FUNCTION_BLOCK AR_CALIBRATE_3P_REF (* Adapter-based 3-point calibration for joysticks/sensors with a center position (Min, Mid, Max), free order like AR_CALIBRATE_3P - reference targets (Y_MIN/Y_MID/Y_MAX) are live AR sockets, persisted via 3 additional AR2 plugs (MIN_REF/MID_REF/MAX_REF), same live-echo pattern as AR_CALIBRATE_SQ_REF/AR_CALIBRATE_2P_REF *)
  (* Standard: 61499-1 *)
  (* Version 1.0, 2026-09-11, Meisterschulen am Ostbahnhof, 3-Punkt-Pendant zu AR_CALIBRATE_2P_REF - fuer Sensoren mit definierter Mittelstellung (z.B. Lenkwinkelsensor: links/geradeaus/rechts). Keine ECC-Reihenfolge-Erzwingung: C_MIN/C_MID/C_MAX speichern unabhaengig, wie AR_CALIBRATE_3P. *)
  (* Version 1.3, 2026-09-21, Franz Höpfinger, Code-Review-Fund (PR #260): xClipping clippte bisher unconditional auf [MIN_REF,MAX_REF], auch wenn nur EIN Punkt kalibriert war - der Partial-Kalibrierung-Fallback (Y.D1 := MIN_REF.DI1/MID_REF.DI1/MAX_REF.DI1) wurde durch den noch unkalibrierten Gegenpart (INI_AR2-Default 0.0) sofort wieder zurueckgeklemmt. Clipping jetzt zusaetzlich an xMinCal AND xMaxCal gegated (MID irrelevant, da Clipping nur gegen MIN_REF/MAX_REF vergleicht). *)
  (* Version 1.2, 2026-09-21, Franz Höpfinger, Bugfix (Franz live am Geraet: 'wenn ich MIN druecke aendert sich der Ausgangswert nicht, erst wenn ich dann auch MID druecke uebernimmt er den MIN wert'): REQ pivotierte bisher immer auf X_MID.DI1, das vor der ersten MID-Kalibrierung beim INI_AR2-Default 0.0 steht - da reale Rohwerte praktisch nie 0.0 sind, war die Bedingung X.D1 < X_MID.DI1 bis zur ersten MID-Kalibrierung permanent falsch und ignorierte MIN/MIN_REF komplett. Neue interne Kalibriert-Flags xMinCal/xMidCal/xMaxCal (latchen TRUE, sobald der jeweilige Rohwert vom INI-Default abweicht - ueberlebt Neustart, da ein echt kalibrierter Punkt nach dem Boot-Restore ebenfalls sofort wieder <> 0.0 ist) lassen REQ bei unvollstaendiger Kalibrierung sauber auf die 1-2-Punkt-Teilloesung bzw. den einzelnen REF-Wert ausweichen, statt mit einem Rohwert-Default von 0.0 zu rechnen. Zusaetzlich: neuer Input xClipping (Default TRUE) macht das bisher fest eingebaute Clipping auf MIN_REF..MAX_REF abschaltbar (FALSE = Extrapolation erlaubt). *)
  (* Version 1.1, 2026-09-18, Franz Höpfinger, C_MIN/C_MID/C_MAX von AX-Sockets (mit [C_x.D1]-Flankenwaechter) auf reine EventInputs umgestellt - jeder echte Aufrufer liefert ohnehin ein atomares Event, der D1-Wert war immer hartcodiert TRUE (via AX_BOOL_TO_X) und der Guard filterte nie etwas. Aufrufer muessen jetzt direkt ein Event statt eines AX-Adapters anschliessen. Siehe AR_CALIBRATE_2P_REF fuer die identische Aenderung. *)
  PACKAGE adapter::Engineering::measurements;
  (* Documentation:
  Formula
   Y = piecewise linear interpolation between (X_MIN,MIN_REF), (X_MID,MID_REF), (X_MAX,MAX_REF), clipped to MIN_REF..MAX_REF unless xClipping = FALSE Partial Calibration (before all 3 points are set)
   Each point is tracked internally (xMinCal/xMidCal/xMaxCal, latched TRUE once its raw value differs from the INI_AR2 default 0.0). Until all three are calibrated, REQ falls back cleanly instead of pivoting on a still-uncalibrated X_MID.DI1 (which would otherwise sit at 0.0 and make the MIN branch permanently unreachable):
    - Only one point calibrated: Y = that point's own REF value (no interpolation possible)
   - Two points calibrated: 2-point line between exactly those two, ignoring the uncalibrated third
   - All three calibrated: full piecewise interpolation as above
   - None calibrated: Y := MID_REF
    Calibration (3-Point, Free Order)
    - Min (C_MIN): Move to minimum, set Y_MIN, trigger C_MIN → X_MIN := X
   - Mid (C_MID): Move to center, set Y_MID, trigger C_MID → X_MID := X
   - Max (C_MAX): Move to maximum, set Y_MAX, trigger C_MAX → X_MAX := X
    Exactly like AR_CALIBRATE_3P: no ECC-enforced order, each point stores independently and can be re-calibrated on its own (e.g. re-trimming a drifted center without touching Min/Max) - unlike a 2-point offset/scale scheme, there is no data dependency between the calibration actions themselves, so an enforced order would only add friction without preventing any actual error.
   Typical use: steering angle sensor
   Min = full lock left, Mid = straight ahead (center), Max = full lock right. MIN_REF/MID_REF/MAX_REF hold the desired calibrated angle values (e.g. -30.0 / 0.0 / 30.0 degrees); X_MIN/X_MID/X_MAX hold whatever raw sensor values were actually measured at those three physical positions.
   Reference Targets (Y_MIN/Y_MID/Y_MAX) are live AR Sockets
   Same live-echo mechanism as AR_CALIBRATE_2P_REF/AR_CALIBRATE_SQ_REF: Y_MIN/Y_MID/Y_MAX are bidirectional AR2 Sockets fed from an external VT/web reader, mirrored out through the AR2 Plugs MIN_REF/MID_REF/MAX_REF for persistence (INI_AR2/NVS_AR2), and echoed back via MIN_REF.EI1/MID_REF.EI1/MAX_REF.EI1 so a boot-restored value shows up on screen without the operator re-entering it.
  *)
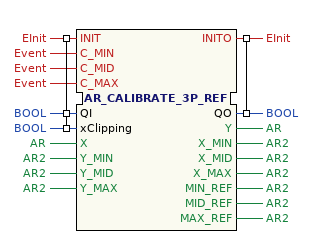
  EVENT_INPUT
    INIT : EInit WITH QI, xClipping; (* Initialization Request *)
    C_MIN; (* Calibrate Min Point - atomarer Trigger *)
    C_MID; (* Calibrate Mid Point (Center) - atomarer Trigger *)
    C_MAX; (* Calibrate Max Point - atomarer Trigger *)
  END_EVENT
  EVENT_OUTPUT
    INITO : EInit WITH QO; (* Initialization Confirm *)
  END_EVENT
  VAR_INPUT
    QI : BOOL; (* Input event qualifier *)
    xClipping : BOOL := TRUE; (* TRUE (Default) = Ausgang wird auf MIN_REF..MAX_REF geklemmt; FALSE = kein Clipping, Extrapolation ueber die Kalibrierpunkte hinaus erlaubt *)
  END_VAR
  VAR_OUTPUT
    QO : BOOL; (* Output event qualifier *)
  END_VAR
  SOCKETS
    X : adapter::types::unidirectional::AR; (* Raw Input *)
    Y_MIN : adapter::types::bidirectional::AR2; (* Target output Y at the Min calibration point - live edit in via EO1/DO1 (Socket-side swap), persisted/restored value echoed back out via EI1/DI1 for VT/web display *)
    Y_MID : adapter::types::bidirectional::AR2; (* Target output Y at the Mid calibration point - live edit in via EO1/DO1 (Socket-side swap), persisted/restored value echoed back out via EI1/DI1 for VT/web display *)
    Y_MAX : adapter::types::bidirectional::AR2; (* Target output Y at the Max calibration point - live edit in via EO1/DO1 (Socket-side swap), persisted/restored value echoed back out via EI1/DI1 for VT/web display *)
  END_SOCKETS
  PLUGS
    Y : adapter::types::unidirectional::AR; (* Calibrated Output *)
    X_MIN : adapter::types::bidirectional::AR2; (* Persisted raw input value at the Min calibration point *)
    X_MID : adapter::types::bidirectional::AR2; (* Persisted raw input value at the Mid (center) calibration point *)
    X_MAX : adapter::types::bidirectional::AR2; (* Persisted raw input value at the Max calibration point *)
    MIN_REF : adapter::types::bidirectional::AR2; (* Persisted Min-point target reference (Y_MIN) *)
    MID_REF : adapter::types::bidirectional::AR2; (* Persisted Mid-point target reference (Y_MID) *)
    MAX_REF : adapter::types::bidirectional::AR2; (* Persisted Max-point target reference (Y_MAX) *)
  END_PLUGS
  VAR
    xMinCal : BOOL := FALSE; (* Latched TRUE sobald X_MIN.DI1 vom INI-Default 0.0 abweicht - MIN wurde mindestens einmal kalibriert (diese Session oder ueber Boot-Restore) *)
    xMidCal : BOOL := FALSE; (* Latched TRUE sobald X_MID.DI1 vom INI-Default 0.0 abweicht - MID wurde mindestens einmal kalibriert (diese Session oder ueber Boot-Restore) *)
    xMaxCal : BOOL := FALSE; (* Latched TRUE sobald X_MAX.DI1 vom INI-Default 0.0 abweicht - MAX wurde mindestens einmal kalibriert (diese Session oder ueber Boot-Restore) *)
  END_VAR
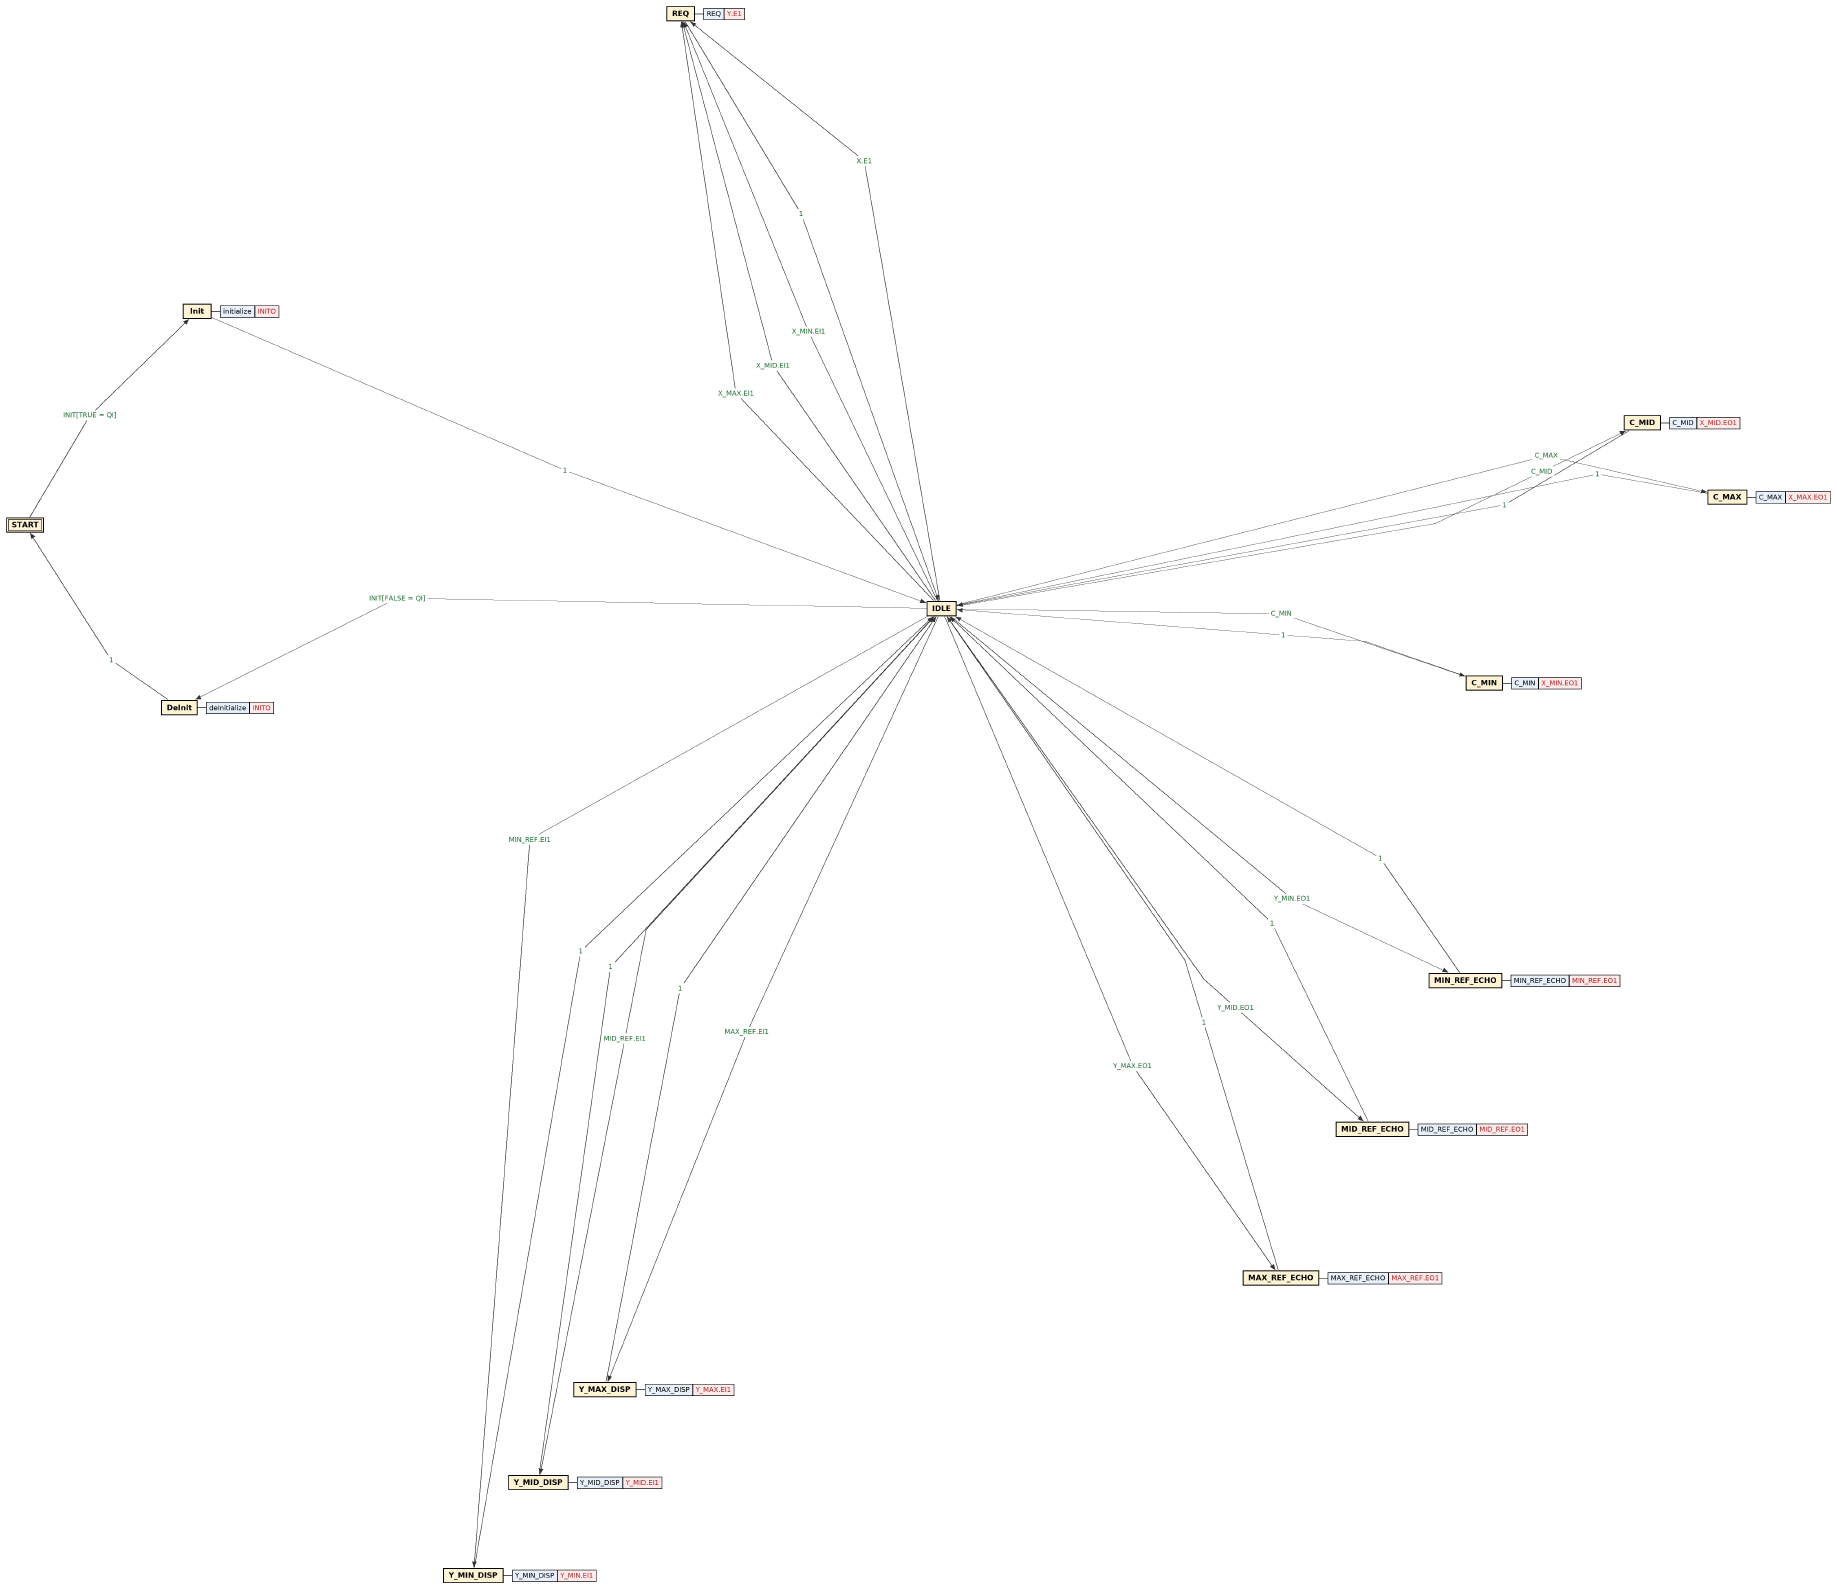
  EC_STATES
    START; (* Initial State *)
    Init : initialize -> INITO; (* Initialization *)
    DeInit : deInitialize -> INITO;
    IDLE;
    REQ : REQ -> Y.E1;
    C_MIN : C_MIN -> X_MIN.EO1;
    C_MID : C_MID -> X_MID.EO1;
    C_MAX : C_MAX -> X_MAX.EO1;
    MIN_REF_ECHO : MIN_REF_ECHO -> MIN_REF.EO1;
    MID_REF_ECHO : MID_REF_ECHO -> MID_REF.EO1;
    MAX_REF_ECHO : MAX_REF_ECHO -> MAX_REF.EO1;
    Y_MIN_DISP : Y_MIN_DISP -> Y_MIN.EI1;
    Y_MID_DISP : Y_MID_DISP -> Y_MID.EI1;
    Y_MAX_DISP : Y_MAX_DISP -> Y_MAX.EI1;
  END_STATES
  EC_TRANSITIONS
    START TO Init := INIT[TRUE = QI];
    DeInit TO START := 1;
    IDLE TO REQ := X.E1;
    REQ TO IDLE := 1;
    IDLE TO C_MIN := C_MIN;
    C_MIN TO IDLE := 1;
    IDLE TO C_MID := C_MID;
    C_MID TO IDLE := 1;
    IDLE TO C_MAX := C_MAX;
    C_MAX TO IDLE := 1;
    IDLE TO REQ := X_MIN.EI1;
    IDLE TO REQ := X_MID.EI1;
    IDLE TO REQ := X_MAX.EI1;
    IDLE TO MIN_REF_ECHO := Y_MIN.EO1;
    MIN_REF_ECHO TO IDLE := 1;
    IDLE TO MID_REF_ECHO := Y_MID.EO1;
    MID_REF_ECHO TO IDLE := 1;
    IDLE TO MAX_REF_ECHO := Y_MAX.EO1;
    MAX_REF_ECHO TO IDLE := 1;
    IDLE TO Y_MIN_DISP := MIN_REF.EI1;
    Y_MIN_DISP TO IDLE := 1;
    IDLE TO Y_MID_DISP := MID_REF.EI1;
    Y_MID_DISP TO IDLE := 1;
    IDLE TO Y_MAX_DISP := MAX_REF.EI1;
    Y_MAX_DISP TO IDLE := 1;
    Init TO IDLE := 1;
    IDLE TO DeInit := INIT[FALSE = QI];
  END_TRANSITIONS
  ALGORITHM initialize IN ST: (* Initialization algorithm *)
QO := QI;
  END_ALGORITHM
  ALGORITHM deInitialize IN ST: (* Normally executed algorithm *)
QO := FALSE;
  END_ALGORITHM
  ALGORITHM REQ IN ST: (* REQ algorithm *)
QO := QI;

IF TRUE = QI THEN
	(* only perform normal operation if QI is true *)

	(* latch "has been calibrated at least once" per point - a never-calibrated point stays
	 * exactly at the INI_AR2 DEFAULT_VALUE (0.0) forever, a real raw sensor value practically
	 * never is; a re-boot restores an already-calibrated point straight back to its non-0.0
	 * persisted value, so the latch stays correctly set across restarts *)
	IF X_MIN.DI1 <> 0.0 THEN xMinCal := TRUE; END_IF;
	IF X_MID.DI1 <> 0.0 THEN xMidCal := TRUE; END_IF;
	IF X_MAX.DI1 <> 0.0 THEN xMaxCal := TRUE; END_IF;

	IF xMinCal AND xMidCal AND xMaxCal THEN
		(* full 3-point piecewise-linear interpolation, exactly as before *)
		IF X.D1 < X_MID.DI1 THEN
			IF X_MID.DI1 > X_MIN.DI1 THEN
				Y.D1 := MIN_REF.DI1 + (X.D1 - X_MIN.DI1) * (MID_REF.DI1 - MIN_REF.DI1) / (X_MID.DI1 - X_MIN.DI1);
			ELSE
				Y.D1 := MIN_REF.DI1;
			END_IF;
		ELSE
			IF X_MAX.DI1 > X_MID.DI1 THEN
				Y.D1 := MID_REF.DI1 + (X.D1 - X_MID.DI1) * (MAX_REF.DI1 - MID_REF.DI1) / (X_MAX.DI1 - X_MID.DI1);
			ELSE
				Y.D1 := MID_REF.DI1;
			END_IF;
		END_IF;
	ELSIF xMinCal AND xMidCal THEN
		(* only MIN+MID calibrated so far - 2-point line between them, MAX not usable yet *)
		IF X_MID.DI1 <> X_MIN.DI1 THEN
			Y.D1 := MIN_REF.DI1 + (X.D1 - X_MIN.DI1) * (MID_REF.DI1 - MIN_REF.DI1) / (X_MID.DI1 - X_MIN.DI1);
		ELSE
			Y.D1 := MIN_REF.DI1;
		END_IF;
	ELSIF xMidCal AND xMaxCal THEN
		(* only MID+MAX calibrated so far - 2-point line between them, MIN not usable yet *)
		IF X_MAX.DI1 <> X_MID.DI1 THEN
			Y.D1 := MID_REF.DI1 + (X.D1 - X_MID.DI1) * (MAX_REF.DI1 - MID_REF.DI1) / (X_MAX.DI1 - X_MID.DI1);
		ELSE
			Y.D1 := MID_REF.DI1;
		END_IF;
	ELSIF xMinCal AND xMaxCal THEN
		(* only MIN+MAX calibrated so far (MID skipped) - direct 2-point line, ignores MID entirely *)
		IF X_MAX.DI1 <> X_MIN.DI1 THEN
			Y.D1 := MIN_REF.DI1 + (X.D1 - X_MIN.DI1) * (MAX_REF.DI1 - MIN_REF.DI1) / (X_MAX.DI1 - X_MIN.DI1);
		ELSE
			Y.D1 := MIN_REF.DI1;
		END_IF;
	ELSIF xMinCal THEN
		Y.D1 := MIN_REF.DI1;
	ELSIF xMidCal THEN
		Y.D1 := MID_REF.DI1;
	ELSIF xMaxCal THEN
		Y.D1 := MAX_REF.DI1;
	ELSE
		(* nothing calibrated yet *)
		Y.D1 := MID_REF.DI1;
	END_IF;

	(* only clip once both outer bounding points are calibrated - otherwise
	 * the still-uncalibrated bound sits at its INI_AR2 default (0.0) and
	 * would clamp the partial-calibration fallback above right back to
	 * garbage. MID is irrelevant here - clipping only ever compares
	 * against MIN_REF/MAX_REF. *)
	IF xClipping AND xMinCal AND xMaxCal THEN
		IF Y.D1 < MIN_REF.DI1 THEN
			Y.D1 := MIN_REF.DI1;
		ELSIF Y.D1 > MAX_REF.DI1 THEN
			Y.D1 := MAX_REF.DI1;
		END_IF;
	END_IF;
END_IF;
  END_ALGORITHM
  ALGORITHM C_MIN IN ST: (* Store current raw input as the Min calibration point - independent, repeatable any time *)
X_MIN.DO1 := X.D1;
  END_ALGORITHM
  ALGORITHM C_MID IN ST: (* Store current raw input as the Mid (center) calibration point - independent, repeatable any time *)
X_MID.DO1 := X.D1;
  END_ALGORITHM
  ALGORITHM C_MAX IN ST: (* Store current raw input as the Max calibration point - independent, repeatable any time *)
X_MAX.DO1 := X.D1;
  END_ALGORITHM
  ALGORITHM MIN_REF_ECHO IN ST: (* Persist live Y_MIN reference to INI *)
MIN_REF.DO1 := Y_MIN.DO1;
  END_ALGORITHM
  ALGORITHM MID_REF_ECHO IN ST: (* Persist live Y_MID reference to INI *)
MID_REF.DO1 := Y_MID.DO1;
  END_ALGORITHM
  ALGORITHM MAX_REF_ECHO IN ST: (* Persist live Y_MAX reference to INI *)
MAX_REF.DO1 := Y_MAX.DO1;
  END_ALGORITHM
  ALGORITHM Y_MIN_DISP IN ST: (* Echo the persisted/restored MIN_REF value back out through Y_MIN for VT/web display (boot and after every change) *)
Y_MIN.DI1 := MIN_REF.DI1;
  END_ALGORITHM
  ALGORITHM Y_MID_DISP IN ST: (* Echo the persisted/restored MID_REF value back out through Y_MID for VT/web display (boot and after every change) *)
Y_MID.DI1 := MID_REF.DI1;
  END_ALGORITHM
  ALGORITHM Y_MAX_DISP IN ST: (* Echo the persisted/restored MAX_REF value back out through Y_MAX for VT/web display (boot and after every change) *)
Y_MAX.DI1 := MAX_REF.DI1;
  END_ALGORITHM
END_FUNCTION_BLOCK
